(* CODESYS project speedometer.export

Project tree, tasks and I/O mapping:
  Device : CODESYS Control Win V3 x64, 3S - Smart Software Solutions GmbH, version 3.5.16.40
    application Application
      libraries: Standard, * (System)
      task MainTask (cyclic, interval t#20ms, priority 1) calls PLC_PRG
      task VISU_TASK (cyclic, interval 100 ms, priority 31) calls VisuElems.Visu_Prg
      program PLC_PRG [CFC]
      visualisation Visualization
*)

// Device/Application/PLC_PRG
PROGRAM PLC_PRG
VAR
	Trykk: BOOL;
	Reset: BOOL;
	Teller: CTU;
	tid1: TON;
	sum: word := 0;
	sum1: WORd := 0;
END_VAR
VAR // added by the converter: edge detectors and wires of the graphical bodies
    _w1 : word;
END_VAR

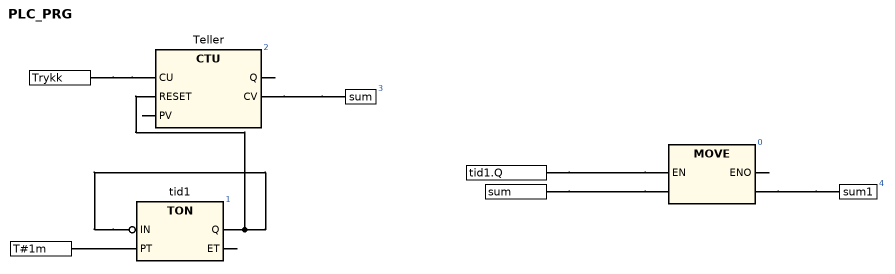
IF tid1.Q THEN _w1 := sum; END_IF
tid1(IN := NOT tid1.Q, PT := T#1m); // TON
Teller(CU := Trykk, RESET := tid1.Q); // CTU
sum := Teller.CV;
sum1 := _w1;

END_PROGRAM

// Device/Application/Visualization
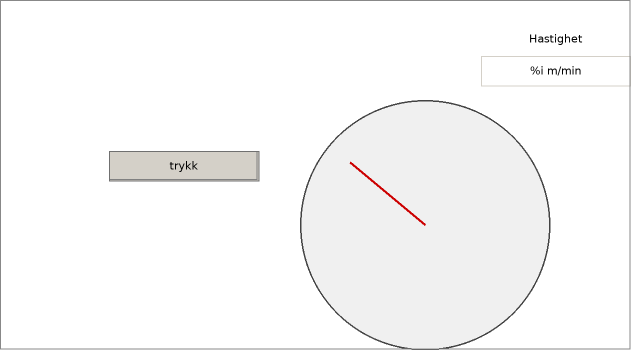
VISUALIZATION Visualization  // 631x350
    Button (109,151 150x30), "trykk"
        tap PLC_PRG.Trykk
    Label (481,24 150x30), "Hastighet"
    Textfield (481,56 150x30), "%i m/min", text variable: PLC_PRG.sum
    Meter90 (300,100 250x250), value: PLC_PRG.sum, style: Meter-Meter90-Gray, scale format: %.1f, scale 0..100
END_VISUALIZATION
